FUNCTION_BLOCK ModbusTCP EXTENDS Modbus
VAR_INPUT
	EN: BOOL;
	{attribute 'TcEncoding':='UTF-8'}
	IP: STRING;
	Port: UINT := 502;
END_VAR
VAR_OUTPUT
	ENO: BOOL;
	Error: BOOL;
END_VAR
VAR
	ModbusMaster: FB_MBReadRegs;
	ModbusMasterWrite: FB_MBWriteRegs;
	{attribute 'TcEncoding':='UTF-8'}
	stMbErrId: STRING;
	aRegisterArray1: ARRAY [1..125] OF WORD;
	aRegisterCoil: ARRAY [1..250] OF BYTE;
	WaitModbusBusy: TON;
	cbRead: INT;
	Param: REFERENCE TO ModbusIo;
	State: INT;
	ReplyTON: LTON;
	LastReadCount: LINT;
END_VAR
VAR PERSISTENT
	tTimeBetweenReads: TIME := T#500MS;
END_VAR

SUPER^();
ENO := EN;
ReplyTON(IN := ReadCount = LastReadCount, PT := LTIME#20S, Q => Error);
LastReadCount := ReadCount;
WaitModbusBusy();
CASE State OF
	0:
		IF EN THEN		
			CurrentIoIndex := 0;
			IF IO[CurrentIoIndex] <> 0 THEN
				State := 5;
			END_IF	
		END_IF
	5:	(* Wait between reads *)
		WaitModbusBusy(IN := TRUE, PT := tTimeBetweenReads, Q=> , ET=> );	
		IF WaitModbusBusy.Q = TRUE THEN
			IF NOT IO[CurrentIoIndex]^.Write THEN
				State := 10;
			ELSE
				State := 110;			
			END_IF
			WaitModbusBusy(IN := FALSE);
		END_IF		
	
	10:
		Param REF= IO[CurrentIoIndex]^; 
		IF NOT Param.EN OR Param.UnitID = 0 THEN
			Param.ValueWord := 0;
			Param.ErrorOUT := FALSE;
			State := 30;
		ELSE
			ModbusMaster(
			sIPAddr:= IP, 
			nTCPPort:= 502, 
			nUnitID:= Param.UnitID, 
			nQuantity:= Param.ParameterCount, 
			nMBAddr:= Param.Register, 
			cbLength:= 2 * Param.ParameterCount, 
			pDestAddr:= ADR(aRegisterArray1), 
			bExecute:= TRUE, 
			tTimeout:= T#1000MS);
			IF  ModbusMaster.bBUSY THEN
				State := State + 10;
			END_IF
		END_IF
	20:
		ModbusMaster();
		IF ModbusMaster.bError THEN
			stMbErrId := concat('Error ', UDINT_TO_STRING(ModbusMaster.nErrId));
			ModbusMaster(bExecute := FALSE);
			Param.ValueWord := 0;
			Param.ErrorOUT := TRUE;
			ErrorCount := ErrorCount + 1;
			ModbusMaster.bExecute:= FALSE;
			State := 30;
		ELSIF NOT ModbusMaster.bBUSY THEN
			ModbusMaster(bExecute := FALSE);
			Param.ValueWord := aRegisterArray1[1];
			Param.ValueWordArray := aRegisterArray1;
			Param.ErrorOUT := FALSE;
			ReadCount := ReadCount + 1;
			ModbusMaster(bExecute:= FALSE);
			State := 30;
		END_IF
	30:
		CurrentIoIndex := CurrentIoIndex + 1;
		IF CurrentIoIndex >= IO_COUNT THEN
			CurrentIoIndex := 0;
		END_IF
		IF IO[CurrentIoIndex] <> 0 THEN
			State := 5;
		ELSE				
			State := 0;
		END_IF
	110:
		Param REF= IO[CurrentIoIndex]^; 
		IF NOT Param.EN OR Param.UnitID = 0 THEN
			Param.ValueWord := 0;
			Param.ErrorOUT := FALSE;
			State := 30;
		ELSE
			aRegisterArray1[1] := Param.ValueWord;
			ModbusMasterWrite(
			sIPAddr:= IP, 
			nTCPPort:= 502, 
			nUnitID:= Param.UnitID, 
			nQuantity:= Param.ParameterCount, 
			nMBAddr:= Param.Register, 
			cbLength:= 2 * Param.ParameterCount, 
			pSrcAddr:= ADR(aRegisterArray1), 
			bExecute:= TRUE, 
			tTimeout:= T#1000MS);
			IF  ModbusMasterWrite.bBUSY THEN
				State := State + 10;
			END_IF
		END_IF
	120:
		ModbusMasterWrite();
		IF ModbusMasterWrite.bError THEN
			stMbErrId := concat('Error ', UDINT_TO_STRING(ModbusMaster.nErrId));
			ModbusMasterWrite(bExecute := FALSE);
			Param.ValueWord := 0;
			Param.ErrorOUT := TRUE;
			ErrorCount := ErrorCount + 1;
			ModbusMasterWrite.bExecute:= FALSE;
			State := 30;
		ELSIF NOT ModbusMasterWrite.bBUSY THEN
			ModbusMasterWrite(bExecute := FALSE);
			Param.ValueWord := aRegisterArray1[1];
			Param.ErrorOUT := FALSE;
			ReadCount := ReadCount + 1;
			ModbusMasterWrite(bExecute:= FALSE);
			State := 30;
		END_IF
		Param.EN := FALSE;
		Param.Write := FALSE;
END_CASE

END_FUNCTION_BLOCK

(* stored: Version 1.1.0.1, ProductVersion 3.1.4024.6
   POU ModbusTCP: Id {c2b301d9-c3e8-4e6e-b0d2-2d7d47081554}, SpecialFunc None *)
